PROGRAM WriteEtherCAT
VAR
	i : INT;
	i2 : INT;
	NetIDString : STRING;
	SymInfo  : ARRAY[1..4]  OF PLC_ReadSymInfoByName;
	SymInd : ARRAY[1..4] OF INT;
	HostFind : FB_GetHostAddrByName;
	COERead : adsread;
	Exec : BOOL;
	destaf : DINT;
END_VAR

//HostFind(sHostName := 'GANTRYKID_1', bExecute := Exec);
//FOR i := 1 TO 4 DO		
//	NetIDString :=INT_TO_STRING(BYTE_TO_INT(main.Kid[i].Address.netId[0]));
//
//	FOR i2 := 1 TO 5 DO NetIDString := CONCAT(Concat(netIDString, '.'), INT_TO_STRING(BYTE_TO_INT(main.Kid[i].Address.netId[i2]))); END_FOR
//SymInfo[i](NetID := NetIDString,  PORT:= main.kid[i].address.port, SymName:= 'TIID^Device 3 (EtherCAT Slave)^Outputs^CurrentPosition_ToMom', Start:=Exec);

	//MAIN.Kid[i].EtherCATWriter();
//END_FOR 	
//COERead(netid:=NetIDString, Port:=851, IDxGRP:=50593872,idxoffs:= 2164260877,Len:=4,DestAddr:=ADR(destaf),read:=Exec);

END_PROGRAM

(* stored: Version 1.1.0.1, ProductVersion 3.1.4022.7
   POU WriteEtherCAT: Id {4b2d570c-56ff-41f3-960a-84c1ae1ecbcf}, SpecialFunc None *)
